Fanuc KAREL source: KD00060.KL

PROGRAM KD00060
%NOLOCKGROUP
VAR
  I: INTEGER
  J: INTEGER
  B: BOOLEAN
  R: REAL
  S: STRING[80]
BEGIN
  CONDITION[1]:
  WHEN DIN[1] = ON DO
    DISABLE CONDITION[1]
  ENDCONDITION
END KD00060
